// TIA Portal V20 export
VAR_GLOBAL   // PLC tag table "ASi Alarm"
   "BW_ASi143 -MCC100 -210KE3 -ConfigErr_Circuit1_Slave(16-31)A" AT %IW66 : Word;
   "BW_ASi143 -MCC100 -210KE3 -ConfigErr_Circuit1_Slave(16-31)B" AT %IW70 : Word;
   "BW_ASi143 -MCC100 -210KE3 -PeriErr_Circuit1_Slave(16-31)A" AT %IW74 : Word;
   "BW_ASi143 -MCC100 -210KE3 -PeriErr_Circuit1_Slave(16-31)B" AT %IW78 : Word;
   "BW_ASi143 -MCC100 -210KE3 -ConfigErr_Circuit2_Slave(0-15)A" AT %IW395 : Word;
   "BW_ASi143 -MCC100 -210KE3 -ConfigErr_Circuit2_Slave(16-31)A" AT %IW397 : Word;
   "BW_ASi143 -MCC100 -210KE3 -ConfigErr_Circuit2_Slave(0-15)B" AT %IW399 : Word;
   "BW_ASi143 -MCC100 -210KE3 -ConfigErr_Circuit2_Slave(16-31)B" AT %IW401 : Word;
   "BW_ASi143 -MCC100 -210KE3 -PeriErr_Circuit2_Slave(0-15)A" AT %IW403 : Word;
   "BW_ASi143 -MCC100 -210KE3 -PeriErr_Circuit2_Slave(16-31)A" AT %IW405 : Word;
   "BW_ASi143 -MCC100 -210KE3 -PeriErr_Circuit2_Slave(0-15)B" AT %IW407 : Word;
   "BW_ASi143 -MCC100 -210KE3 -PeriErr_Circuit2_Slave(16-31)B" AT %IW409 : Word;
   "BW_ASi143 -MCC100 -210KE3 -ConfigErr_Circuit1_Slave(0-15)A" AT %IW64 : Word;
   "BW_ASi143 -MCC100 -210KE3 -ConfigErr_Circuit1_Slave(0-15)B" AT %IW68 : Word;
   "BW_ASi143 -MCC100 -210KE3 -PeriErr_Circuit1_Slave(0-15)A" AT %IW72 : Word;
   "BW_ASi143 -MCC100 -210KE3 -PeriErr_Circuit1_Slave(0-15)B" AT %IW76 : Word;
   "BW_ASi200 -MCC300 -210KE3 -ConfigErr_Circuit1_Slave(0-15)A" AT %IW513 : Word;
   "BW_ASi200 -MCC300 -210KE3 -ConfigErr_Circuit1_Slave(16-31)A" AT %IW515 : Word;
   "BW_ASi200 -MCC300 -210KE3 -ConfigErr_Circuit1_Slave(0-15)B" AT %IW517 : Word;
   "BW_ASi200 -MCC300 -210KE3 -ConfigErr_Circuit1_Slave(16-31)B" AT %IW519 : Word;
   "BW_ASi200 -MCC300 -210KE3 -PeriErr_Circuit1_Slave(0-15)A" AT %IW521 : Word;
   "BW_ASi200 -MCC300 -210KE3 -PeriErr_Circuit1_Slave(16-31)A" AT %IW523 : Word;
   "BW_ASi200 -MCC300 -210KE3 -PeriErr_Circuit1_Slave(0-15)B" AT %IW525 : Word;
   "BW_ASi200 -MCC300 -210KE3 -PeriErr_Circuit1_Slave(16-31)B" AT %IW527 : Word;
   "BW_ASi200 -MCC300 -210KE3 -ConfigErr_Circuit2_Slave(0-15)A" AT %IW529 : Word;
   "BW_ASi200 -MCC300 -210KE3 -ConfigErr_Circuit2_Slave(16-31)A" AT %IW531 : Word;
   "BW_ASi200 -MCC300 -210KE3 -ConfigErr_Circuit2_Slave(0-15)B" AT %IW533 : Word;
   "BW_ASi200 -MCC300 -210KE3 -ConfigErr_Circuit2_Slave(16-31)B" AT %IW535 : Word;
   "BW_ASi200 -MCC300 -210KE3 -PeriErr_Circuit2_Slave(0-15)A" AT %IW537 : Word;
   "BW_ASi200 -MCC300 -210KE3 -PeriErr_Circuit2_Slave(16-31)A" AT %IW539 : Word;
   "BW_ASi200 -MCC300 -210KE3 -PeriErr_Circuit2_Slave(0-15)B" AT %IW541 : Word;
   "BW_ASi200 -MCC300 -210KE3 -PeriErr_Circuit2_Slave(16-31)B" AT %IW543 : Word;
END_VAR
